ABB RAPID module: LoaderPositions.mod

MODULE LoaderPositions

    CONST orient LOADERPICKUPANGLE := [0.29789,-0.24355,0.63677,0.66819];
    CONST orient LOADERDROPANGLE := [0.55589,0.67049,0.04049,-0.48968];
    CONST robtarget TRAY1 := [ [0, 399.3, 672.1],LOADERPICKUPANGLE, [0,0,-1,1], [9E9,9E9,9E9,9E9,9E9,9E9] ];
    CONST robtarget TRAY2 := [ [0, 402, 576.7],LOADERPICKUPANGLE, [0,0,-1,1], [9E9,9E9,9E9,9E9,9E9,9E9] ];
    CONST robtarget TRAY3 := [ [0, 410.8, 477.1],LOADERPICKUPANGLE, [0,0,-1,1], [9E9,9E9,9E9,9E9,9E9,9E9] ];
    CONST robtarget TRAY4 := [ [0, 414.9, 377.9],LOADERPICKUPANGLE, [0,0,-1,1], [9E9,9E9,9E9,9E9,9E9,9E9] ];
    CONST robtarget TRAY5 := [ [0, 420.6, 278.6],LOADERPICKUPANGLE, [0,0,-1,1], [9E9,9E9,9E9,9E9,9E9,9E9] ];
    CONST robtarget TRAY6 := [ [0, 424.6, 179.8],LOADERPICKUPANGLE, [0,0,-1,1], [9E9,9E9,9E9,9E9,9E9,9E9] ];
    CONST robtarget LOADERDROP := [ [-124.2, -178.4, 500],LOADERDROPANGLE, [0,0,-1,1], [9E9,9E9,9E9,9E9,9E9,9E9] ];

ENDMODULE
